Staubli VAL3: Instruction.dtx

public bool bIsTraj
public string sPath
public string sID
public bool bUseOnPoint
public num nIndex
